// Mitsubishi GX Works2 project: IELET2103_Datalab2   PLC: FX2N/FX2NC
// IELET2103_Datalab2

// task Task_01 (event TRUE, interval 0, priority 31): Oppgav1Figur2_ST

PROGRAM Oppgave1
(* structured ladder/FBD written out as ST: instructions are called as NAME(EN, inputs, outputs); _pN, _eN, _tN stand for wires *)
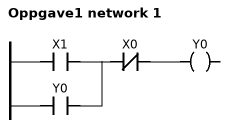
(* network 1 *)
Y0 := (X1 OR Y0) AND NOT X0;
END_PROGRAM

PROGRAM Oppgave1_IL
// body in language c0 not rendered
END_PROGRAM

PROGRAM Oppgave1_ST
Y0 := (X1 OR Y0) AND NOT X0;
END_PROGRAM

PROGRAM Oppgave1Figur2_Ladder
(* structured ladder/FBD written out as ST: instructions are called as NAME(EN, inputs, outputs); _pN, _eN, _tN stand for wires *)
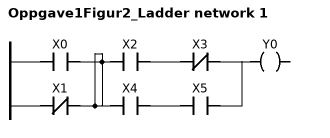
(* network 1 *)
_p1 := X0 OR (NOT X1);
Y0 := (_p1 AND X2 AND NOT X3) OR (_p1 AND X4 AND X5);
END_PROGRAM

PROGRAM Oppgav1Figur2_ST
Y0 :=  (X0 OR NOT X1) AND ((X2 AND NOT X3) OR (X4 AND X5));
END_PROGRAM

PROGRAM Oppgave1Figur2_IL
// body in language c0 not rendered
END_PROGRAM
